PROGRAM FB_Mode

VAR_INPUT
	iStatusPowerOn:				BOOL; //true if the machine is powered on
	iStatusMotivePowerOn:		BOOL; //true if the machine motive power is on (drives, air, etc)

	iManualMode:				BOOL; //manual button
	iAutoMode:					BOOL; //auto button
	iStartAutoCycle:			BOOL; //start auto cycle button
	iSemiAutoMode:				BOOL; //semi auto button
	iContCycle:					BOOL; //continuous cycle mode
	iSingleCycle:				BOOL; //single cycle mode
	iHome:						BOOL;  //station is at HOME
	iFault:						BOOL;
	iDryCycleMode:				BOOL; //station in dry cycle mode



	iIsStationSelected: BOOL; //is the current station selected?
END_VAR
	
	
VAR
	
END_VAR

VAR_OUTPUT
	qManualMode: BOOL;
	qAutoMode: BOOL;
	qAutoCycling: BOOL;
	qSemiAuto: BOOL; 
	qContCycle: BOOL; //machine is in continous cycle mode
	qSingleCycle: BOOL; //machine is in single cycle mode, auto cycle will stop when HOME is reached
	qDryCycle: BOOL; //machine will function as normal but with no part present sensors feedback



	qModeState: INT; //value feedback for HMI


END_VAR

VAR_IN_OUT
	stationState:typeStationMode;
	
END_VAR
VAR // added by the converter: edge detectors and wires of the graphical bodies
    _rt1, _rt2, _rt3, _rt4, _rt5 : R_TRIG;
    _w1, _w2, _w3 : BOOL;
END_VAR

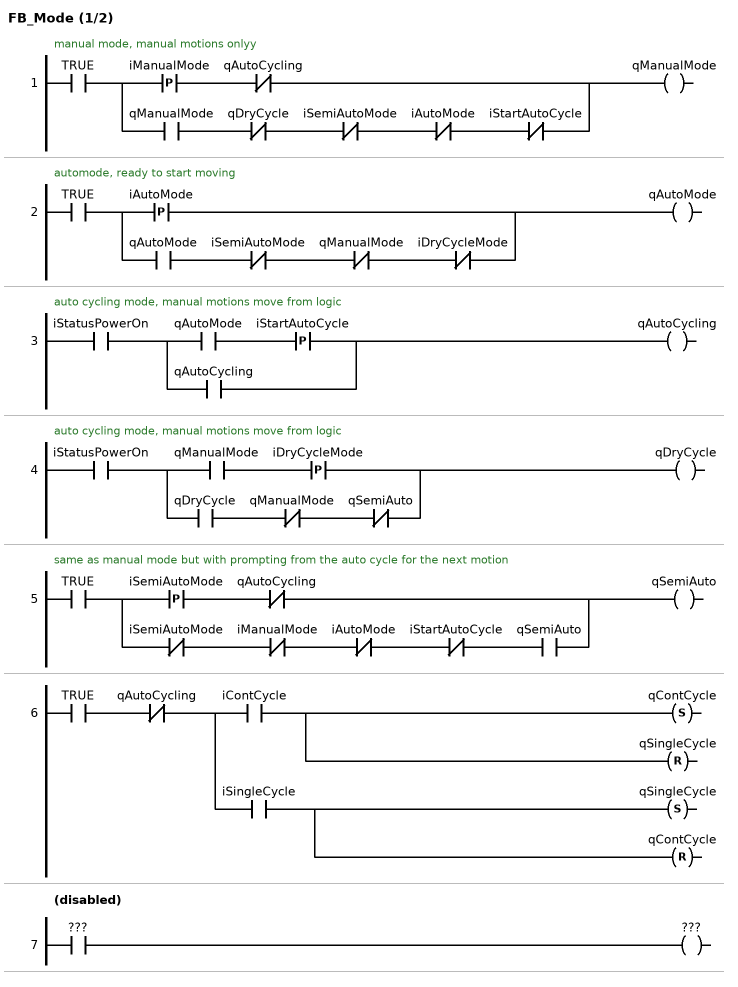
// NETWORK 1
// manual mode, manual motions onlyy
_rt1(CLK := iManualMode);
qManualMode := TRUE AND (_rt1.Q AND NOT qAutoCycling OR qManualMode AND NOT qDryCycle AND NOT iSemiAutoMode AND NOT iAutoMode AND NOT iStartAutoCycle);

// NETWORK 2
// automode, ready to start moving
_rt2(CLK := iAutoMode);
qAutoMode := TRUE AND (_rt2.Q OR qAutoMode AND NOT iSemiAutoMode AND NOT qManualMode AND NOT iDryCycleMode);

// NETWORK 3
// auto cycling mode, manual motions move from logic
_rt3(CLK := iStartAutoCycle);
qAutoCycling := iStatusPowerOn AND (qAutoMode AND _rt3.Q OR qAutoCycling);

// NETWORK 4
// auto cycling mode, manual motions move from logic
_rt4(CLK := iDryCycleMode);
qDryCycle := iStatusPowerOn AND (qManualMode AND _rt4.Q OR qDryCycle AND NOT qManualMode AND NOT qSemiAuto);

// NETWORK 5
// same as manual mode but with prompting from the auto cycle for the next motion
_rt5(CLK := iSemiAutoMode);
qSemiAuto := TRUE AND (_rt5.Q AND NOT qAutoCycling OR NOT iSemiAutoMode AND NOT iManualMode AND NOT iAutoMode AND NOT iStartAutoCycle AND qSemiAuto);

// NETWORK 6
_w1 := TRUE AND NOT qAutoCycling;
_w2 := _w1 AND iContCycle;
qContCycle S= _w2;
qSingleCycle R= _w2;
_w3 := _w1 AND iSingleCycle;
qSingleCycle S= _w3;
qContCycle R= _w3;

// NETWORK 7 (disabled)
// ??? := ???;

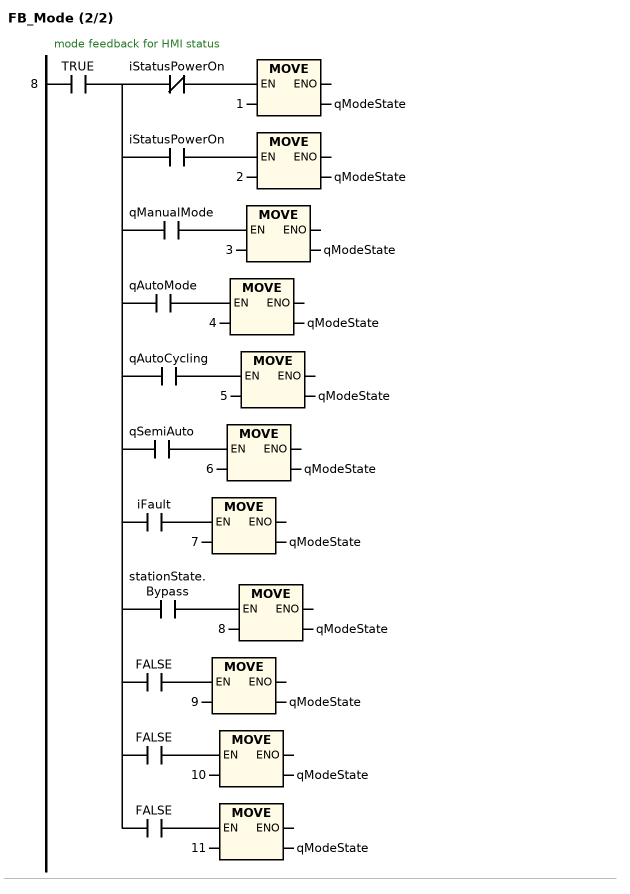
// NETWORK 8
// mode feedback for HMI status
IF TRUE AND NOT iStatusPowerOn THEN qModeState := 1; END_IF
IF TRUE AND iStatusPowerOn THEN qModeState := 2; END_IF
IF TRUE AND qManualMode THEN qModeState := 3; END_IF
IF TRUE AND qAutoMode THEN qModeState := 4; END_IF
IF TRUE AND qAutoCycling THEN qModeState := 5; END_IF
IF TRUE AND qSemiAuto THEN qModeState := 6; END_IF
IF TRUE AND iFault THEN qModeState := 7; END_IF
IF TRUE AND stationState.Bypass THEN qModeState := 8; END_IF
IF TRUE AND FALSE THEN qModeState := 9; END_IF
IF TRUE AND FALSE THEN qModeState := 10; END_IF
IF TRUE AND FALSE THEN qModeState := 11; END_IF

END_PROGRAM

(* stored: Version 1.1.0.1, ProductVersion 3.1.4024.12
   POU FB_Mode: Id {ce08c7f1-a47e-41ce-a12a-5019455503c9}, SpecialFunc None *)
